{attribute 'qualified_only'}
VAR_GLOBAL CONSTANT
	ANGLE_STATIONARY : LREAL := 999;
	
	NOT_ON_RAIL : INT := 0;
	RAIL_LEFT : INT := 1;
	RAIL_RIGHT : INT := 2;
	
END_VAR

(* stored: Version 1.1.0.1, ProductVersion 3.1.4026.13
   GVL CollisionDetection: Id {41ff17ea-9a34-4626-85aa-508c49f790c3} *)
